INTERFACE I_GraphVisitor EXTENDS I_MetadataVisitor, I_InputPortVisitor, I_OutputPortVisitor, I_ContentVisitor, I_ParameterVisitor, I_ErrorVisitor, I_ExtensionVisitor, I_NodeVisitor

METHOD VisitGraph
VAR_INPUT
	VisitingGraph : I_Graph;
END_VAR
END_METHOD

END_INTERFACE

(* stored: Version 1.1.0.1, ProductVersion 3.1.4024.12
   Itf I_GraphVisitor: Id {3beaad77-f9b4-0e1e-36c4-b261c862bbf6}
   Method VisitGraph: Id {57ece38e-dc27-051d-27f8-98538b3ae4ff} *)
